FUNCTION_BLOCK INTERNAL FB_Year EXTENDS FB_Object IMPLEMENTS I_SeasonControl, I_CyclicTask
VAR
    fbSeasonStateMachine:   FB_SeasonStateMachine;
    fbWinter:               FB_Winter(THIS^.fbSeasonStateMachine, THIS^);
    fbSpring:               FB_Spring(THIS^.fbSeasonStateMachine, THIS^);
    fbSummer:               FB_Summer(THIS^.fbSeasonStateMachine, THIS^);
    fbAutumn:               FB_Autumn(THIS^.fbSeasonStateMachine, THIS^);

    nCounter:               UDINT;
    nModVal:                UDINT := 500;
END_VAR

METHOD ChangeToSummerTyres
VAR_INPUT
END_VAR
THIS^.CurrentState().ChangeToSummerTyres();
END_METHOD

METHOD ChangeToWinterTyres
VAR_INPUT
END_VAR
THIS^.CurrentState().ChangeToWinterTyres();
END_METHOD

METHOD CurrentState : I_SeasonState
__QUERYINTERFACE(THIS^.fbSeasonStateMachine.ipState, CurrentState);
END_METHOD

METHOD FB_init : BOOL
VAR_INPUT
    bInitRetains:           BOOL; // if TRUE, the retain variables are initialized (warm start / cold start)
    bInCopyCode:            BOOL;  // if TRUE, the instance afterwards gets moved into the copy code (online change)
END_VAR
THIS^.fbSeasonStateMachine.SetState(THIS^.StateSummer);
THIS^.CurrentState().ChangeToSummerTyres();
END_METHOD

METHOD NextSeason
VAR_INPUT
END_VAR
THIS^.fbSeasonStateMachine.NextSeason();
END_METHOD

METHOD Run
VAR_INPUT
END_VAR
THIS^.nCounter := THIS^.nCounter + 1;
THIS^.fbSeasonStateMachine.Run();
END_METHOD

PROPERTY StateAutumn : I_State
GET
StateAutumn := THIS^.fbAutumn;
END_GET
END_PROPERTY

PROPERTY StateSpring : I_State
GET
StateSpring := THIS^.fbSpring;
END_GET
END_PROPERTY

PROPERTY StateSummer : I_State
GET
StateSummer := THIS^.fbSummer;
END_GET
END_PROPERTY

PROPERTY StateWinter : I_State
GET
StateWinter := THIS^.fbWinter;
END_GET
END_PROPERTY

END_FUNCTION_BLOCK

(* stored: Version 1.1.0.1, ProductVersion 3.1.4024.12
   POU FB_Year: Id {fe655ad5-7059-0731-0988-2edb45df25ec}, SpecialFunc None
   Folder Properties: Id {ee3573fd-0509-051c-0602-8171ec30d53c}
   Method ChangeToSummerTyres: Id {70ebc0db-cf84-0f7e-3fab-533965158ac1}
   Method ChangeToWinterTyres: Id {20add137-020c-0490-2dee-a5aae9b1e602}
   Method CurrentState: Id {9dde5f23-25e2-0c5b-1d72-636cd789ec37}
   Method FB_init: Id {903d718b-fbcd-043f-2b03-d4b812d5787f}
   Method NextSeason: Id {cc87e7e1-d903-0057-1226-7c1055a0d405}
   Method Run: Id {652743c6-ccfc-020d-276e-cddc5e1bb354}
   Property StateAutumn: Id {2e1d0bde-c684-0c08-3f60-61b11c35adc8}
   Get Get: Id {6c74ae4c-0fa2-0cde-15ed-402bfd0b4100}
   Property StateSpring: Id {374866af-9ff1-094a-0ef4-a5727719ca68}
   Get Get: Id {ef19480a-5df6-0247-1038-2002c554b65a}
   Property StateSummer: Id {cddc9c39-53d3-09d9-2b73-00dcb11b7762}
   Get Get: Id {4ca04d3b-f233-09d9-3400-c2e2b3ec87a1}
   Property StateWinter: Id {6b7932ed-be28-0650-3513-fca56ba90efa}
   Get Get: Id {8e64ce48-6662-0c98-1586-05362dd69e90} *)
